Staubli VAL3: OnEvent17.pgx

program OnEvent17()
  local bool l_bBool
begin
  //-----------------------------------------------------------------------
  //Header begin
  //LasMAN3.7
  //Description of program
  //
  //Input parameters
  //
  //Output paramaters
  //Example
  //  call OnEvent1()
  //History
  //  Creation : 2013-06-23  y.ye@staubli.com
  //Header end
  //-----------------------------------------------------------------------
  resetMotion()
  call UI:Control_YesNO("确定替换空白的调试文件吗?",l_bBool)
  if l_bBool
    call TxtFile:SaveNewProduct(l_bBool)

  endIf
  DataBase:nInterfaceType=9
end
